TYPE ST_UAMethodCall_AdsReadDeviceInfoRes :
STRUCT
	nNumberOfOutputArguments	: UDINT;
	nReserved					: ARRAY [1..4] OF BYTE; // padding
	stOutputArgInfo				: ARRAY [1..4] OF ST_UAMethodArgInfo;
	stDeviceInfo				: ST_DeviceInfo;
END_STRUCT
END_TYPE

(* stored: Version 1.1.0.1, ProductVersion 3.1.4022.6
   DUT ST_UAMethodCall_AdsReadDeviceInfoRes: Id {b2d2973b-86ab-43fa-8ec6-eda5eb31effc} *)
